# B&R Automation Studio project MotionTestBenchMaster (part 59)

#### LiftMoveMngt_Doser.st
```iecst
ACTION LiftMoveMngt_Doser:

	VAR_DOS_Lift_State.DevicesGeneralAlarm := MMF[205].OUT_DriveFault OR MMF[205].OUT_OverloadFault OR MMF[206].OUT_DriveFault OR
												MMF[206].OUT_OverloadFault OR _205MEF.OUT_Alarm OR _206MEF.OUT_Alarm;

	VAR_DOS_Lift_State.CmdProductionHeight.Sp	:= HMI_PAR_1._215; //[ml]
	VAR_DOS_Lift_State.CmdCipHeight.Sp			:= 145.0; //[ml]

	VAR_DOS_PistonVolume_ml := 145.0; 	(*ml*)  //Max Volume [ml]
	VAR_DOS_PistonVolume_mm := 180.0;	(*mm*)  //Max height of recipe [mm]

	FbLCRLimScal_ml_mm(
	x1 := 0.0, 		(*ml*)
	y1 := 0.0, 		(*mm*)
	x2 := VAR_DOS_PistonVolume_ml, 	(*ml*)
	y2 := VAR_DOS_PistonVolume_mm,	(*mm*)
	);

	FbLCRLimScal_mm_ml(
	x1 := 0.0, 		(*mm*)
	y1 := 0.0, 		(*ml*)
	x2 := VAR_DOS_PistonVolume_mm, 	(*mm*)
	y2 := VAR_DOS_PistonVolume_ml,	(*ml*)
	);

	IF (VAR_DOS_ModePositionRequest AND (VAR_DOS_ModeWait AND NOT COP.DataOut.RcpActive)) THEN
		VAR_DOS_MMF205.SpActual[mm]	:= 200.0; //DEFINE-> Hema Valves "free" - Cam horizontal
		VAR_DOS_MMF206.SpActual[mm]	:= 200.0;
	ELSIF ((VAR_DOS_ModePositionRequest AND (VAR_DOS_ModeProduction OR VAR_DOS_FMDProductionFillerOnly)) OR (HMI_DOS_LiftPosition.Value = 1)) THEN
		VAR_DOS_MMF205.SpActual[ml] := MIN(VAR_DOS_Lift_State.CmdProductionHeight.Sp,VAR_DOS_PistonVolume_ml);
		FbLCRLimScal_ml_mm.x 		:= VAR_DOS_MMF205.SpActual[ml];
		VAR_DOS_MMF205.SpActual[mm]	:= FbLCRLimScal_ml_mm.y;
		VAR_DOS_MMF206.SpActual[mm]	:= 0.0;
	ELSIF ((VAR_DOS_ModePositionRequest AND (VAR_DOS_ModeCip OR VAR_DOS_ModeRinse)) OR (HMI_DOS_LiftPosition.Value = 3)) THEN
		VAR_DOS_MMF205.SpActual[ml] := MIN(VAR_DOS_Lift_State.CmdCipHeight.Sp,VAR_DOS_PistonVolume_ml);
		FbLCRLimScal_ml_mm.x 		:= VAR_DOS_MMF205.SpActual[ml];
		VAR_DOS_MMF205.SpActual[mm]	:= FbLCRLimScal_ml_mm.y;
		VAR_DOS_MMF206.SpActual[mm]	:= 0.0;
	ELSIF ((VAR_DOS_ModePositionRequest AND VAR_DOS_ModeCop AND COP.DataOut.DoserPositioningReq) OR (HMI_DOS_LiftPosition.Value = 2)) THEN
		VAR_DOS_MMF205.SpActual[mm] := 322.0; //High sensor height _215DSF  Define in Test
		VAR_DOS_MMF205.SpActual[ml] := 0;
		VAR_DOS_MMF206.SpActual[mm]	:= 323.0;
	ELSIF HMI_DOS_SS2P[SS2P_DOS_ProbeAdjustment].ON THEN
		VAR_DOS_MMF205.SpActual[mm] := 0.0;
		VAR_DOS_MMF206.SpActual[mm]	:= VAR_DOS_MMF205.SpActual[mm]; //--> Define in Test _205MEF.IN_Delta and _206MEF.IN_Delta
	ELSE
		VAR_DOS_MMF205.SpActual[mm] := 0.0;
		VAR_DOS_MMF205.SpActual[ml] := 0.0;
		VAR_DOS_MMF206.SpActual[mm] := 0.0;
	END_IF

	memset(ADR(VAR_DOS_LiftMMF205SeqMem), 0, SIZEOF(VAR_DOS_LiftMMF205SeqMem));
	memset(ADR(VAR_DOS_LiftMMF206SeqMem), 0, SIZEOF(VAR_DOS_LiftMMF206SeqMem));
	HMI_DOS_PB[PB_DOS_Up].Enable		:= FALSE;
	HMI_DOS_PB[PB_DOS_Down].Enable		:= FALSE;
	_211CPF.IN_AutoCnd 					:= FALSE;
	IF EDGEPOS(VAR_DOS_Lift_State.DevicesGeneralAlarm) THEN
		VAR_DOS_LiftStepMem := VAR_DOS_LiftMoveStep;
	END_IF

	IF EDGENEG(VAR_DOS_ModeWait) OR NOT HMI_DOS_LiftPosition.Enable THEN
		HMI_DOS_LiftPosition.Value := 0;
	END_IF

	IF EDGEPOS(VAR_DOS_FMDPositionRequest) THEN
		VAR_DOS_SeqPositionReached := FALSE;
	END_IF

	//*******************************************************************************************************************************************
	CASE VAR_DOS_LiftMoveStep OF
		DSR_LiftSystemOff:
			HMI_DOS_Lift_State.Sequencer.TextBar[0].IndexNr		:= 0;
			HMI_DOS_Lift_State.Sequencer.TextBar[0].IndexText	:= 0;

			VAR_DOS_LiftMMF205SeqMem.Position.ActualSp	:= VAR_DOS_MMF205.SpActual[ml]; //[ml]

			IF HMI_DOS_SS2P[SS2P_DOS_SelLiftMan].ON THEN
				VAR_DOS_LiftMoveStep := DSR_Manual;
			ELSIF HMI_DOS_SS2P[SS2P_DOS_ProbeAdjustment].ON THEN
				VAR_DOS_LiftMoveStep := DSR_ProbeZeroReq;
			ELSIF (VAR_DOS_ModePositionRequest AND NOT VAR_DOS_SeqPositionReached AND VAR_DOS_ModeWait AND NOT COP.DataOut.RcpActive) THEN
				VAR_DOS_LiftMoveStep := DSR_PosMMF206ToMMF205;
			ELSIF ((VAR_DOS_ModeCop AND COP.DataOut.DoserPositioningReq AND NOT VAR_DOS_SeqPositionReached) OR (EDGEPOS(HMI_DOS_PB[PB_CmdLiftMotorStart].ON) AND HMI_DOS_LiftPosition.Value = 2)) THEN
				VAR_DOS_LiftMoveStep := DSR_PosMMF206ToMMF205;
			ELSIF (((VAR_DOS_ModeProduction OR VAR_DOS_FMDProductionFillerOnly) AND VAR_DOS_ModePositionRequest AND NOT VAR_DOS_SeqPositionReached) OR (EDGEPOS(HMI_DOS_PB[PB_CmdLiftMotorStart].ON) AND HMI_DOS_LiftPosition.Value = 1))THEN
				VAR_DOS_LiftMoveStep := DSR_DosingReq;
			ELSIF (((VAR_DOS_ModeCip OR VAR_DOS_ModeRinse) AND VAR_DOS_ModePositionRequest AND NOT VAR_DOS_SeqPositionReached) OR (EDGEPOS(HMI_DOS_PB[PB_CmdLiftMotorStart].ON) AND HMI_DOS_LiftPosition.Value = 3)) THEN
				VAR_DOS_LiftMoveStep := DSR_DosingReq;
			END_IF

		DSR_ProbeZeroReq:
			HMI_DOS_Lift_State.Sequencer.TextBar[0].IndexNr		:= 1;
			HMI_DOS_Lift_State.Sequencer.TextBar[0].IndexText	:= 1;

			VAR_DOS_LiftMoveStep := DSR_ProbeZeroLowPos;
			IF NOT HMI_DOS_SS2P[SS2P_DOS_ProbeAdjustment].ON THEN
				VAR_DOS_LiftMoveStep := DSR_LiftSystemOff;
			END_IF

		DSR_ProbeZeroLowPos:
			HMI_DOS_Lift_State.Sequencer.TextBar[0].IndexNr		:= 2;
			HMI_DOS_Lift_State.Sequencer.TextBar[0].IndexText	:= 2;

			IF NOT VAR_DOS_Lift_State.DevicesGeneralAlarm THEN

				IF ((VAR_DOS_MMF205.PosActual[mm] <= VAR_DOS_MMF205.SpActual[mm]) OR VAR_DOS_MMF205.SensorLowPos OR (VAR_DOS_MMF205.PosActual[mm] < VAR_DOS_MMF206.PosActual[mm] - 5.0)) THEN
					VAR_DOS_LiftMMF205SeqMem.LiftMotor.Dwn := FALSE;
				ELSIF VAR_DOS_MMF205.SpActual[mm] <= VAR_DOS_MMF205.PosActual[mm] THEN
					VAR_DOS_LiftMMF205SeqMem.LiftMotor.Dwn := TRUE;
				END_IF

				IF ((VAR_DOS_MMF206.PosActual[mm] <= VAR_DOS_MMF206.SpActual[mm]) OR VAR_DOS_MMF206.SensorLowPos OR (VAR_DOS_MMF206.PosActual[mm] <= VAR_DOS_MMF205.PosActual[mm] - VAR_DOS_PistonVolume_mm)) THEN
					VAR_DOS_LiftMMF206SeqMem.LiftMotor.Dwn := FALSE;
				ELSIF ((VAR_DOS_MMF206.PosActual[mm] >= VAR_DOS_MMF205.SpActual[mm]) OR (VAR_DOS_MMF206.PosActual[mm] >= VAR_DOS_MMF206.SpActual[mm] AND VAR_DOS_MMF205.PosReached)) (*mm*)THEN
					VAR_DOS_LiftMMF206SeqMem.LiftMotor.Dwn := TRUE;
				END_IF

				IF VAR_DOS_LiftMMF205SeqMem.LiftMotor.Dwn THEN
					IF VAR_DOS_MMF205.SensorMaxVol THEN
						VAR_DOS_LiftMMF205SeqMem.Sensor.SensorMaxVolWaitOff := TRUE;
					ELSIF NOT VAR_DOS_MMF205.SensorLowPos THEN
						VAR_DOS_LiftMMF205SeqMem.Sensor.SensorLowPosWaitOn := TRUE;
					END_IF
				END_IF

				IF VAR_DOS_LiftMMF206SeqMem.LiftMotor.Dwn THEN
					IF NOT VAR_DOS_MMF206.SensorLowPos THEN
						VAR_DOS_LiftMMF206SeqMem.Sensor.SensorLowPosWaitOn := TRUE;
					END_IF
				END_IF

				IF NOT VAR_DOS_LiftMMF205SeqMem.LiftMotor.Dwn AND NOT VAR_DOS_LiftMMF206SeqMem.LiftMotor.Dwn THEN
					VAR_DOS_LiftMoveStep := DSR_ProbeZeroDisengSensLow;
				END_IF

				IF NOT HMI_DOS_SS2P[SS2P_DOS_ProbeAdjustment].ON THEN
					VAR_DOS_LiftMoveStep := DSR_LiftSystemOff;
				END_IF

			END_IF

		DSR_ProbeZeroDisengSensLow:
			HMI_DOS_Lift_State.Sequencer.TextBar[0].IndexNr		:= 3;
			HMI_DOS_Lift_State.Sequencer.TextBar[0].IndexText	:= 3;

			IF NOT VAR_DOS_Lift_State.DevicesGeneralAlarm THEN
				VAR_DOS_LiftMMF205SeqMem.LiftMotor.Up := VAR_DOS_MMF205.SensorLowPos;
				VAR_DOS_LiftMMF206SeqMem.LiftMotor.Up := VAR_DOS_MMF206.SensorLowPos;

				VAR_DOS_LiftMMF205SeqMem.Sensor.SensorLowPosWaitOff := VAR_DOS_LiftMMF205SeqMem.LiftMotor.Up AND VAR_DOS_MMF205.SensorLowPos;
				VAR_DOS_LiftMMF206SeqMem.Sensor.SensorLowPosWaitOff := VAR_DOS_LiftMMF206SeqMem.LiftMotor.Up AND VAR_DOS_MMF206.SensorLowPos;

				IF NOT VAR_DOS_LiftMMF205SeqMem.LiftMotor.Up AND NOT VAR_DOS_LiftMMF206SeqMem.LiftMotor.Up THEN
					VAR_DOS_LiftMoveStep := DSR_ProbeZeroWaitSensLowPos;
				END_IF

				IF NOT HMI_DOS_SS2P[SS2P_DOS_ProbeAdjustment].ON THEN
					VAR_DOS_LiftMoveStep := DSR_LiftSystemOff;
				END_IF
			END_IF

		DSR_ProbeZeroWaitSensLowPos:
			HMI_DOS_Lift_State.Sequencer.TextBar[0].IndexNr		:= 4;
			HMI_DOS_Lift_State.Sequencer.TextBar[0].IndexText	:= 4;

			IF NOT VAR_DOS_Lift_State.DevicesGeneralAlarm THEN
				VAR_DOS_LiftMMF205SeqMem.LiftMotor.Dwn := NOT VAR_DOS_MMF205.SensorLowPos;
				VAR_DOS_LiftMMF206SeqMem.LiftMotor.Dwn := NOT VAR_DOS_MMF206.SensorLowPos;

				VAR_DOS_LiftMMF205SeqMem.Sensor.SensorLowPosWaitOff := VAR_DOS_LiftMMF205SeqMem.LiftMotor.Up AND NOT VAR_DOS_MMF205.SensorLowPos;
				VAR_DOS_LiftMMF206SeqMem.Sensor.SensorLowPosWaitOff := VAR_DOS_LiftMMF206SeqMem.LiftMotor.Up AND NOT VAR_DOS_MMF206.SensorLowPos;

				IF NOT VAR_DOS_LiftMMF205SeqMem.LiftMotor.Dwn AND NOT VAR_DOS_LiftMMF206SeqMem.LiftMotor.Dwn THEN
					VAR_DOS_MMF205.PosValid := FALSE;
					VAR_DOS_MMF206.PosValid := FALSE;
					Delta_205MEF			:= 0.0;
					Delta_206MEF			:= 0.0;
					VAR_DOS_LiftMoveStep	:= DSR_ProbeZeroDone;
				END_IF
			END_IF

			IF NOT HMI_DOS_SS2P[SS2P_DOS_ProbeAdjustment].ON THEN
				VAR_DOS_LiftMoveStep := DSR_LiftSystemOff;
			END_IF

		DSR_ProbeZeroDone:
			HMI_DOS_Lift_State.Sequencer.TextBar[0].IndexNr		:= 5;
			HMI_DOS_Lift_State.Sequencer.TextBar[0].IndexText	:= 5;

			IF NOT VAR_DOS_Lift_State.DevicesGeneralAlarm THEN
				IF NOT VAR_DOS_MMF205.PosValid THEN
					Delta_205MEF			:= -(_205MEF.OUT_ActValue + Delta_205MEF) + 0.5;
					VAR_DOS_MMF205.PosValid := TRUE;
				END_IF

				IF NOT VAR_DOS_MMF206.PosValid THEN
					Delta_206MEF 		:= -(_206MEF.OUT_ActValue + Delta_206MEF) + 0.5;
					VAR_DOS_MMF206.PosValid := TRUE;
				END_IF
			END_IF

			IF VAR_DOS_MMF205.PosValid AND VAR_DOS_MMF206.PosValid THEN
				HMI_DOS_SS2P[SS2P_DOS_ProbeAdjustment].ON := FALSE;
				VAR_DOS_LiftMoveStep					  := DSR_LiftSystemOff;
			END_IF

		DSR_PosMMF206ToMMF205:
			HMI_DOS_Lift_State.Sequencer.TextBar[0].IndexNr		:= 10;
			HMI_DOS_Lift_State.Sequencer.TextBar[0].IndexText	:= 10;
			VAR_DOS_LiftMMF205SeqMem.Position.ActualSp	:= VAR_DOS_MMF205.SpActual[ml]; //[ml]
			VAR_DOS_SeqPositionReached	:= FALSE;

			IF NOT VAR_DOS_Lift_State.DevicesGeneralAlarm THEN
				IF VAR_DOS_ModeCop THEN
					VAR_DOS_LiftMMF206SeqMem.LiftMotor.Up := (VAR_DOS_MMF206.PosActual[mm] < VAR_DOS_MMF205.PosActual[mm]);
					IF NOT VAR_DOS_LiftMMF206SeqMem.LiftMotor.Up THEN
						VAR_DOS_LiftMoveStep := DSR_UpMMF205andMMF206;
					END_IF
				ELSIF VAR_DOS_MMF205.SpActual[mm] >= VAR_DOS_MMF205.PosActual[mm] THEN
					VAR_DOS_LiftMMF206SeqMem.LiftMotor.Up := VAR_DOS_MMF206.PosActual[mm] < VAR_DOS_MMF205.PosActual[mm];
					IF NOT VAR_DOS_LiftMMF206SeqMem.LiftMotor.Up THEN
						VAR_DOS_LiftMoveStep := DSR_UpMMF205andMMF206;
					END_IF
				END_IF
			ELSE
				VAR_DOS_LiftMoveStep := DSR_Fault;
			END_IF

		DSR_UpMMF205andMMF206:
			HMI_DOS_Lift_State.Sequencer.TextBar[0].IndexNr		:= 11;
			HMI_DOS_Lift_State.Sequencer.TextBar[0].IndexText	:= 11;

			VAR_DOS_LiftMMF205SeqMem.Position.ActualSp	:= VAR_DOS_MMF205.SpActual[ml]; //[ml]

			IF EDGEPOS(HMI_DOS_PB[PB_CmdLiftMotorStop].ON) THEN
				VAR_DOS_LiftMoveStep := DSR_LiftSystemOff;
			END_IF

			IF NOT VAR_DOS_Lift_State.DevicesGeneralAlarm THEN

				IF ((VAR_DOS_MMF205.PosActual[mm] > VAR_DOS_MMF205.SpActual[mm]) OR VAR_DOS_MMF205.SensorHighPos OR (VAR_DOS_MMF205.PosActual[mm] > VAR_DOS_MMF206.PosActual[mm] + VAR_DOS_PistonVolume_mm)) THEN
					VAR_DOS_LiftMMF205SeqMem.LiftMotor.Up := FALSE;
				ELSIF VAR_DOS_MMF205.SpActual[mm] >= VAR_DOS_MMF205.PosActual[mm] THEN
					VAR_DOS_LiftMMF205SeqMem.LiftMotor.Up := TRUE;
				END_IF

				IF ((VAR_DOS_MMF206.PosActual[mm] > VAR_DOS_MMF206.SpActual[mm]) OR VAR_DOS_MMF206.SensorHighPos OR (VAR_DOS_MMF206.PosActual[mm] > VAR_DOS_MMF205.PosActual[mm] + 5.0)) THEN
					VAR_DOS_LiftMMF206SeqMem.LiftMotor.Up := FALSE;
				ELSIF VAR_DOS_MMF206.PosActual[mm] <= VAR_DOS_MMF206.SpActual[mm] THEN //CHECK
					VAR_DOS_LiftMMF206SeqMem.LiftMotor.Up := TRUE;
				END_IF

				IF NOT VAR_DOS_LiftMMF205SeqMem.LiftMotor.Up THEN
					VAR_DOS_MMF205.PosReached := TRUE;
				ELSE
					VAR_DOS_MMF205.PosReached := FALSE;
				END_IF

				IF NOT VAR_DOS_LiftMMF206SeqMem.LiftMotor.Up THEN
					VAR_DOS_MMF206.PosReached := TRUE;
				ELSE
					VAR_DOS_MMF206.PosReached := FALSE;
				END_IF

				IF ((VAR_DOS_ModeCop AND COP.DataOut.DoserPositioningReq) OR (VAR_DOS_ModeWait AND (HMI_DOS_LiftPosition.Value = 2))) THEN
					IF VAR_DOS_MMF206.PosReached AND VAR_DOS_MMF205.PosReached AND VAR_DOS_MMF205.SensorHighPos AND VAR_DOS_MMF206.SensorHighPos THEN
						VAR_DOS_LiftMoveStep := DSR_CopPosReached;
					END_IF
				ELSE
					VAR_DOS_LiftMoveStep := DSR_LiftSystemOff;
				END_IF
			ELSE
				VAR_DOS_LiftMoveStep := DSR_Fault;
			END_IF

		DSR_DwnMMF205andMMF206:
			HMI_DOS_Lift_State.Sequencer.TextBar[0].IndexNr		:= 12;
			HMI_DOS_Lift_State.Sequencer.TextBar[0].IndexText	:= 12;

			VAR_DOS_LiftMMF205SeqMem.Position.ActualSp	:= VAR_DOS_MMF205.SpActual[ml]; //[ml]

			IF EDGEPOS(HMI_DOS_PB[PB_CmdLiftMotorStop].ON) THEN
				VAR_DOS_LiftMoveStep := DSR_LiftSystemOff;
			END_IF

			IF NOT VAR_DOS_Lift_State.DevicesGeneralAlarm THEN

				IF ((VAR_DOS_MMF205.PosActual[mm] < VAR_DOS_MMF205.SpActual[mm]) OR VAR_DOS_MMF205.SensorLowPos OR (VAR_DOS_MMF205.PosActual[mm] < VAR_DOS_MMF206.PosActual[mm] - 5.0)) THEN
					VAR_DOS_LiftMMF205SeqMem.LiftMotor.Dwn := FALSE;
				ELSIF VAR_DOS_MMF205.SpActual[mm] <= VAR_DOS_MMF205.PosActual[mm] THEN
					VAR_DOS_LiftMMF205SeqMem.LiftMotor.Dwn := TRUE;
				END_IF

				IF ((VAR_DOS_MMF206.PosActual[mm] < VAR_DOS_MMF206.SpActual[mm]) OR VAR_DOS_MMF206.SensorLowPos OR (VAR_DOS_MMF206.PosActual[mm] <= VAR_DOS_MMF205.PosActual[mm] - VAR_DOS_PistonVolume_mm)) THEN
					VAR_DOS_LiftMMF206SeqMem.LiftMotor.Dwn := FALSE;
				ELSIF ((VAR_DOS_MMF206.PosActual[mm] >= VAR_DOS_MMF205.SpActual[mm]) OR (VAR_DOS_MMF206.PosActual[mm] >= VAR_DOS_MMF206.SpActual[mm])) (*mm*)THEN
					VAR_DOS_LiftMMF206SeqMem.LiftMotor.Dwn := TRUE;
					END_IF

				IF NOT VAR_DOS_LiftMMF205SeqMem.LiftMotor.Dwn THEN
					VAR_DOS_MMF205.PosReached := TRUE;
				ELSE
					VAR_DOS_MMF205.PosReached := FALSE;
				END_IF

				IF NOT VAR_DOS_LiftMMF206SeqMem.LiftMotor.Dwn THEN
					VAR_DOS_MMF206.PosReached := TRUE;
				ELSE
					VAR_DOS_MMF206.PosReached := FALSE;
				END_IF

				IF (VAR_DOS_ModeCop AND COP.DataOut.DoserPositioningReq) OR (VAR_DOS_ModeWait AND HMI_DOS_LiftPosition.Value = 2) THEN
					IF VAR_DOS_MMF206.PosReached AND VAR_DOS_MMF206.SensorHighPos AND VAR_DOS_MMF205.SensorHighPos THEN
						VAR_DOS_LiftMoveStep := DSR_CopPosReached;
					END_IF
				ELSIF (VAR_DOS_ModeProduction OR VAR_DOS_FMDProductionFillerOnly) OR (VAR_DOS_ModeWait AND HMI_DOS_LiftPosition.Value = 1)THEN
					IF VAR_DOS_MMF206.PosReached AND VAR_DOS_MMF206.SensorLowPos THEN
						VAR_DOS_LiftMoveStep := DSR_DosingActive;
					END_IF
				ELSIF (VAR_DOS_ModeCip OR VAR_DOS_ModeRinse) OR (VAR_DOS_ModeWait AND HMI_DOS_LiftPosition.Value = 3) THEN
					IF VAR_DOS_MMF206.PosReached AND VAR_DOS_MMF206.SensorLowPos THEN
						VAR_DOS_LiftMoveStep := DSR_DosingActive;
					END_IF
				ELSE
					VAR_DOS_LiftMoveStep := DSR_LiftSystemOff;
				END_IF
			ELSE
				VAR_DOS_LiftMoveStep := DSR_Fault;
			END_IF

		DSR_CopPosReached:
			HMI_DOS_Lift_State.Sequencer.TextBar[0].IndexNr		:= 6;
			HMI_DOS_Lift_State.Sequencer.TextBar[0].IndexText	:= 6;

			VAR_DOS_LiftMMF205SeqMem.Position.ActualSp	:= VAR_DOS_MMF205.SpActual[ml]; //[ml]

			_211CPF.IN_AutoCnd := COP.DataOut.DoserPositioningReq AND VAR_DOS_MMF205.SensorHighPos AND VAR_DOS_MMF206.SensorHighPos;

			VAR_DOS_SeqPositionReached := _210DSX.OUT;

			IF NOT COP.DataOut.DoserPositioningReq AND _211DSX.OUT THEN
				VAR_DOS_LiftMoveStep := DSR_LiftSystemOff;
			END_IF

		DSR_DosingReq:
			HMI_DOS_Lift_State.Sequencer.TextBar[0].IndexNr		:= 7;
			IF VAR_DOS_ModeCip THEN
				HMI_DOS_Lift_State.Sequencer.TextBar[0].IndexText	:= 15;//CIP
			ELSIF VAR_DOS_ModeProduction THEN
				HMI_DOS_Lift_State.Sequencer.TextBar[0].IndexText	:= 7;//PRODUCTION
			END_IF
			VAR_DOS_LiftMMF205SeqMem.Position.ActualSp	:= VAR_DOS_MMF205.SpActual[ml]; //[ml]
			VAR_DOS_SeqPositionReached	:= FALSE;

			IF NOT VAR_DOS_MMF206.SensorLowPos THEN
				VAR_DOS_LiftMoveStep := DSR_DwnMMF205andMMF206;
			ELSE
				VAR_DOS_LiftMoveStep := DSR_DosingActive;
			END_IF

		DSR_DosingActive:
			HMI_DOS_Lift_State.Sequencer.TextBar[0].IndexNr		:= 8;
			HMI_DOS_Lift_State.Sequencer.TextBar[0].IndexText	:= 8;

			VAR_DOS_LiftMMF205SeqMem.Position.ActualSp	:= VAR_DOS_MMF205.SpActual[ml]; //[ml]

			IF EDGEPOS(HMI_DOS_PB[PB_CmdLiftMotorStop].ON) THEN
				VAR_DOS_LiftMoveStep := DSR_LiftSystemOff;
			END_IF

			IF NOT VAR_DOS_Lift_State.DevicesGeneralAlarm THEN

				IF ((VAR_DOS_MMF205.PosActual[mm] > VAR_DOS_MMF205.SpActual[mm]) OR VAR_DOS_MMF205.SensorHighPos OR VAR_DOS_MMF205.SensorMaxVol OR (VAR_DOS_MMF205.PosActual[mm] > VAR_DOS_MMF206.PosActual[mm] + VAR_DOS_PistonVolume_mm)) THEN
					VAR_DOS_LiftMMF205SeqMem.LiftMotor.Up := FALSE;
				ELSIF VAR_DOS_MMF205.SpActual[mm] - 0.5 >= VAR_DOS_MMF205.PosActual[mm] THEN
					VAR_DOS_LiftMMF205SeqMem.LiftMotor.Up := TRUE;
				END_IF

				IF ((VAR_DOS_MMF205.PosActual[mm] < VAR_DOS_MMF205.SpActual[mm]) OR VAR_DOS_MMF205.SensorLowPos) THEN
					VAR_DOS_LiftMMF205SeqMem.LiftMotor.Dwn := FALSE;
				ELSIF VAR_DOS_MMF205.SpActual[mm] + 0.5 <= VAR_DOS_MMF205.PosActual[mm] THEN
					VAR_DOS_LiftMMF205SeqMem.LiftMotor.Dwn := TRUE;
				END_IF

				IF (NOT VAR_DOS_LiftMMF205SeqMem.LiftMotor.Up AND NOT VAR_DOS_LiftMMF205SeqMem.LiftMotor.Dwn) THEN
					VAR_DOS_MMF205.PosReached := TRUE;
				ELSE
					VAR_DOS_MMF205.PosReached := FALSE;
				END_IF

				VAR_DOS_MMF206.PosReached	:= VAR_DOS_MMF206.SensorLowPos;

				VAR_DOS_SeqPositionReached	:= VAR_DOS_MMF205.PosReached AND VAR_DOS_MMF206.PosReached;

				IF VAR_DOS_SeqPositionReached THEN
					VAR_DOS_LiftMoveStep := DSR_LiftSystemOff;
				END_IF
			ELSE
				VAR_DOS_LiftMoveStep := DSR_Fault;
			END_IF

		DSR_Manual:
			HMI_DOS_Lift_State.Sequencer.TextBar[0].IndexNr		:= 9;
			HMI_DOS_Lift_State.Sequencer.TextBar[0].IndexText	:= 9;

			VAR_DOS_LiftMMF205SeqMem.Position.ActualSp	:= VAR_DOS_MMF205.SpActual[ml]; //[ml]

			IF NOT VAR_DOS_Lift_State.DevicesGeneralAlarm THEN
				IF HMI_DOS_SS2P[SS2P_DOS_ManualMMF205].LampON AND NOT VAR_DOS_MMF205.SensorHighPos AND VAR_DOS_MMF205.PosActual[mm] <= VAR_DOS_MMF206.PosActual[mm] + VAR_DOS_PistonVolume_mm THEN
					HMI_DOS_PB[PB_DOS_Up].Enable := TRUE;
					VAR_DOS_LiftMMF205SeqMem.LiftMotor.Up := HMI_DOS_PB[PB_DOS_Up].LampON;
				ELSIF HMI_DOS_SS2P[SS2P_DOS_ManualMMF206].LampON AND NOT VAR_DOS_MMF206.SensorHighPos AND VAR_DOS_MMF206.PosActual[mm] <= VAR_DOS_MMF205.PosActual[mm] THEN
					HMI_DOS_PB[PB_DOS_Up].Enable := TRUE;
					VAR_DOS_LiftMMF206SeqMem.LiftMotor.Up := HMI_DOS_PB[PB_DOS_Up].LampON;
				END_IF

				IF HMI_DOS_SS2P[SS2P_DOS_ManualMMF205].LampON AND NOT VAR_DOS_MMF205.SensorLowPos AND VAR_DOS_MMF205.PosActual[mm] >= VAR_DOS_MMF206.PosActual[mm] - 10.0 THEN
					HMI_DOS_PB[PB_DOS_Down].Enable := TRUE;
					VAR_DOS_LiftMMF205SeqMem.LiftMotor.Dwn := HMI_DOS_PB[PB_DOS_Down].LampON;
				ELSIF HMI_DOS_SS2P[SS2P_DOS_ManualMMF206].LampON AND NOT VAR_DOS_MMF206.SensorLowPos AND VAR_DOS_MMF206.PosActual[mm] >= VAR_DOS_MMF205.PosActual[mm] - VAR_DOS_PistonVolume_mm THEN
					HMI_DOS_PB[PB_DOS_Down].Enable := TRUE;
					VAR_DOS_LiftMMF206SeqMem.LiftMotor.Dwn := HMI_DOS_PB[PB_DOS_Down].LampON;
				END_IF
			END_IF

			IF NOT HMI_DOS_SS2P[SS2P_DOS_SelLiftMan].ON THEN
				VAR_DOS_LiftMoveStep := DSR_LiftSystemOff;
			END_IF

		DSR_Fault:
			HMI_DOS_Lift_State.Sequencer.TextBar[0].IndexNr	:= 13;
			HMI_DOS_Lift_State.Sequencer.TextBar[0].IndexText 	:= 13;

			VAR_DOS_SeqPositionReached	:= FALSE;

			VAR_DOS_LiftMMF205SeqMem.Position.ActualSp	:= VAR_DOS_MMF205.SpActual[ml] * BOOL_TO_REAL(VAR_DOS_ModePositionRequest);
			IF NOT VAR_DOS_Lift_State.DevicesGeneralAlarm THEN
				VAR_DOS_LiftMoveStep := VAR_DOS_LiftStepMem;
			END_IF

	END_CASE
	//******************************************************************************************************************************************

	MMF[205].IN_AutoCnd		:= (VAR_DOS_LiftMMF205SeqMem.LiftMotor.Up AND NOT VAR_DOS_MMF205.SensorHighPos) OR
	(VAR_DOS_LiftMMF205SeqMem.LiftMotor.Dwn AND NOT VAR_DOS_MMF205.SensorLowPos);
	MMF[205].IN_Reverse		:= VAR_DOS_LiftMMF205SeqMem.LiftMotor.Dwn AND MMF[205].IN_AutoCnd;

	MMF[206].IN_AutoCnd		:= (VAR_DOS_LiftMMF206SeqMem.LiftMotor.Up AND NOT VAR_DOS_MMF206.SensorHighPos) OR
	(VAR_DOS_LiftMMF206SeqMem.LiftMotor.Dwn AND NOT VAR_DOS_MMF206.SensorLowPos);
	MMF[206].IN_Reverse		:= VAR_DOS_LiftMMF206SeqMem.LiftMotor.Dwn AND MMF[206].IN_AutoCnd;

	_215DSF.IN_WaitOn	:= VAR_DOS_LiftMMF205SeqMem.Sensor.SensorHighPosWaitOn;
	_215DSF.IN_WaitOff	:= VAR_DOS_LiftMMF205SeqMem.Sensor.SensorHighPosWaitOff;

	_216DSF.IN_WaitOn	:= VAR_DOS_LiftMMF206SeqMem.Sensor.SensorHighPosWaitOn;
	_216DSF.IN_WaitOff	:= VAR_DOS_LiftMMF206SeqMem.Sensor.SensorHighPosWaitOff;
	_217DSF.IN_WaitOn	:= VAR_DOS_LiftMMF206SeqMem.Sensor.SensorLowPosWaitOn;
	_217DSF.IN_WaitOff	:= VAR_DOS_LiftMMF206SeqMem.Sensor.SensorLowPosWaitOff;

	VAR_DOS_MMF205.SensorHighPos := _215DSF.OUT AND NOT _212DSF.OUT AND NOT _213DSF.OUT;
	VAR_DOS_MMF205.SensorMaxVol  := NOT _212DSF.OUT AND _213DSF.OUT;
	VAR_DOS_MMF205.SensorLowPos	 := NOT _213DSF.OUT AND NOT _215DSF.OUT AND _212DSF.OUT;
	VAR_DOS_MMF205.PosActual[mm] := _205MEF.OUT_ActValue;
	FbLCRLimScal_mm_ml.x		 := VAR_DOS_MMF205.PosActual[mm];
	VAR_DOS_MMF205.PosActual[ml] := FbLCRLimScal_mm_ml.y;

	VAR_DOS_MMF206.SensorHighPos := _216DSF.OUT AND NOT _217DSF.OUT;
	VAR_DOS_MMF206.SensorLowPos  := _217DSF.OUT AND NOT _216DSF.OUT;
	VAR_DOS_MMF206.PosActual[mm] := _206MEF.OUT_ActValue;

	IF _205MEF.OUT_Alarm AND MMF[205].OUT_InOperation THEN
		VAR_DOS_MMF205.PosValid := FALSE;
	END_IF
	IF _206MEF.OUT_Alarm AND MMF[206].OUT_InOperation THEN
		VAR_DOS_MMF206.PosValid := FALSE;
	END_IF

	END_ACTION
```

#### DOS_DataOut.st
```iecst
ACTION DOS_DataOut:

	//SEQUENCE
	DOS.DataOut.WaitMode		:= VAR_DOS_ModeWait;
	DOS.DataOut.ProdMode		:= VAR_DOS_ModeProduction;
	DOS.DataOut.CipMode 		:= VAR_DOS_ModeCip;
	DOS.DataOut.RinseMode		:= VAR_DOS_ModeRinse;
	DOS.DataOut.CopMode			:= VAR_DOS_ModeCop AND VAR_DOS_SeqPositionReached;
	DOS.DataOut.DrainMode		:= VAR_DOS_ModeDrain;
	DOS.DataOut.CopAfterCipReq  := VAR_DOS_SEQ.Mem.CopAfterCipRequest;
	DOS.DataOut.CopRunning		:= VAR_DOS_StepCopRunning;

	//SIGNALS INTERCHANGE
	DOS.DataOut.FillingProd		:= VAR_DOS_StepProdProducing OR VAR_DOS_StepProdEndProduction;
	DOS.DataOut.CommandToValve	:= VAR_DOS_SEQ.Mem.ValveOpening OR COP.DataOut.RcpActive;
	DOS.DataOut.ProductRequest	:= VAR_DOS_SEQ.ITC.PROD_ProductRequest; //PULP REQ
	DOS.DataOut.ProductionEnd	:= VAR_DOS_SEQ.ITC.PROD_EndProductionCompleted;
	DOS.DataOut.ReadyForHeating := VAR_DOS_SEQ.ITC.PROD_ReadyForHeating; //HOT WATER REQ
	DOS.DataOut.DoserInTemperature := TTJ[203].OUT_SpReached;
	DOS.DataOut.DoserFull		:= LTJ[203].OUT_SpReached AND VAR_DOS_StepProdHeating; //ONLY IN START UP ?
	DOS.DataOut.AVJ201Open		:= AVJ[201].OUT_OpenedFiltered;
	DOS.DataOut.DoserEmpty		:= VAR_DOS_TankEmpted;
	DOS.DataOut.RecoveryEnd		:= VAR_DOS_SEQ.ITC.PROD_ProductRecoveryEnd;

	DOS.DataOut.CipConditionOk	:= VAR_DOS_ModeCip AND VAR_DOS_SeqPositionReached AND NOT VAR_DOS_SeqCipStopAlarm AND TTJ[203].OUT_SpReached; //CIP SOLUT REQ AND CIP SOLUTION RETURN
	DOS.DataOut.CipSolutionReq	:= VAR_DOS_SEQ.ITC.CIP_CleaningRequest;
	DOS.DataOut.CipAlarm		:= VAR_DOS_SeqCipStopAlarm; //VALUTA
	DOS.DataOut.CipRecovery		:= VAR_DOS_StepCipRecovery AND IO_AVJ[216].DI_Opened AND AVJ[217].OUT (*AND IO_AVJ[218].DI_Opened*) AND PPJ[202].OUT_InOperation;
	DOS.DataOut.CipRecoveryEnd  := VAR_DOS_SEQ.ITC.CIP_ChangeEnded;
	DOS.DataOut.CipSystemFlooded := VAR_DOS_SEQ.ITC.CIP_FloodingEnded;
	DOS.DataOut.CipDrainEnd		:= VAR_DOS_SEQ.ITC.CIP_DrainEnded;
	DOS.DataOut.CipLevelReached := LTJ[203].OUT_SpReached AND VAR_DOS_ModeCip; //Allo step 73 A2 aspetta che tutti i partner siano a livelloCIP e poi chiude tutto in loop

	DOS.DataOut.RinseReq		:= VAR_DOS_SEQ.ITC.CIP_RinseRunning;
	DOS.DataOut.RinseEnd		:= VAR_DOS_SEQ.ITC.CIP_RinseEnded;
	DOS.DataOut.RinseAfterProdReq := VAR_DOS_SEQ.ITC.PROD_WaterRequestAfterProd;
	DOS.DataOut.RinseAfterProdEnd := VAR_DOS_SEQ.ITC.CIP_RinseEnded;

	DOS.DataOut.EjectionRequest	:= VAR_DOS_RejectExpulsionRequest;
	DOS.DataOut.HotWaterReq		:= VAR_DOS_StepCipDraining; //At the end of the CIP, rinse of hot water

	DOS.DataOut.NecessaryBottleEndProd := VAR_DOS_ProdEndNecessaryBottle;

	//FIX SPEED
	DOS.DataOut.FixSpeedRequest := (VAR_DOS_ModeCip AND NOT TNK.DataOut.CipMode) OR VAR_DOS_ModeCop OR (VAR_DOS_ModeRinse AND NOT TNK.DataOut.RinseMode);

	IF VAR_DOS_ModeCip OR VAR_DOS_ModeRinse THEN
		DOS.DataOut.FixSpeedValue := HMI_PAM_3._631;
	ELSIF VAR_DOS_FMDCop THEN
		DOS.DataOut.FixSpeedValue := HMI_PAM_3._632;
	END_IF

	//MOTION
	DOS.DataOut.MachineStart			:= VAR_DOS_SEQ.Mem.MachineStart;
	DOS.DataOut.MachineStop				:= VAR_DOS_SEQ.Mem.MachineStop;
	DOS.DataOut.DoserExcluded 			:= VAR_DOS_MemDoserByPassed;
	DOS.DataOut.DoserIncluded			:= VAR_DOS_MemDoserIncluded;
	DOS.DataOut.ByPassed				:= GNS.DataOut.DosByPassed;
	DOS.DataOut.PhasingWithDos			:= VAR_DOS_PhasingWithDos;
	DOS.DataOut.PhasingWithoutDos			:= VAR_DOS_PhasingWithoutDos;

	IF OPS.DataOut.FlrModeSelectorAdjustment AND NOT MNM.DataOut.MachineRunning THEN //machine running non so se serve
		DOS.DataOut.AxisDisableRequest		:= FALSE;
		DOS.DataOut.RunOnlyHemaAxisRequest := FALSE;
	ELSE
		DOS.DataOut.AxisDisableRequest		:= VAR_DOS_MemDoserAxisOff;
		DOS.DataOut.AxisEnableRequest		:= VAR_DOS_MemDoserAxisOn;
		DOS.DataOut.RunOnlyHemaAxisRequest  := VAR_DOS_MemFillerAxisOffReq AND NOT TNK.DataOut.StartCipRinser;
		DOS.DataOut.RunRinserHemaAxisRequest := VAR_DOS_MemFillerAxisOffReq AND RNS.DataOut.RunWithHemaReq;
	END_IF

	DOS.DataOut.StepCounterRequest		:= VAR_DOS_SEQ.Mem.LapsCounter;

	DOS.DataOut.PositionReached 		:= VAR_DOS_SeqPositionReached;

	//FILLER SELECTION ENABLE
	DOS.DataOut.FillerProdStartEnable	:= VAR_DOS_ModeWait OR VAR_DOS_ModeProduction;
	DOS.DataOut.FillerCipStartEnable	:= VAR_DOS_ModeWait OR (VAR_DOS_ModeCip AND VAR_DOS_StepCipFillerStartEnable);
	DOS.DataOut.FillerRinseStartEnable	:= VAR_DOS_ModeWait OR VAR_DOS_ModeRinse; //VALUTARE: AND NOT VAR_DOS_StepRinseInExecution)
END_ACTION
```

#### DOS_DataOutFlavor.st
```iecst
ACTION DOS_DataOutFlavor:
	//FLAVOR DOSER
	DOS.DataOut.ProdMode 	:= REAL_TO_BOOL(HMI_PAR_1._005) AND TNK.DataOut.ProdMode;
	DOS.DataOut.CipMode 	:= DosFlr.CipReady OR DosFlr.CipRunning;
	DOS.DataOut.AromePodReq := REAL_TO_BOOL(HMI_PAR_1._005) AND TNK.DataOut.ProdMode;
	DOS.DataOut.MachineStart := DosFlr.RotationRequest;

	IF DOS.DataOut.AromePodReq AND NOT ALR[3100].Active AND DosFlr.PrimingCycleProgress THEN
		DOS.DataOut.FixSpeedRequest 		:= TRUE;
		DOS.DataOut.FixSpeedValue 			:= CFG_MC.Movements.MachineMaxSpeed;
	ELSIF DosFlr.RotationRequest AND NOT ALR[3100].Active AND DOS.DataOut.CipMode THEN
		DOS.DataOut.FixSpeedRequest 		:= TRUE;
		DOS.DataOut.FixSpeedValue 			:= MIN(20000, CFG_MC.Movements.MachineMaxSpeed *0.7);
	ELSIF DosFlr.SampleCycleInProgress THEN
		DOS.DataOut.FixSpeedRequest		 	:= TRUE;
		DOS.DataOut.FixSpeedValue 			:= MIN(10000, CFG_MC.Movements.MachineMaxSpeed *0.5);
	ELSE
		DOS.DataOut.FixSpeedRequest		 	:= FALSE;
		DOS.DataOut.FixSpeedValue 			:= 0;
	END_IF
END_ACTION
```

#### DOS_HMI.st
```iecst
ACTION DOS_HMI:
	VAR_DOS_MemPBStart			:= FALSE;
	VAR_DOS_MemPBStop			:= FALSE;
	VAR_DOS_MemPBAbort			:= FALSE;
	VAR_DOS_MemPBSkipForward	:= FALSE;

	IF NOT HMI_SS2P[SS2P_HMI_SelEnable].ON THEN
		HMI_DOS_SS2P[SS2P_DOS_SelLiftMan].ON := FALSE;
	END_IF

	//SS2P
	//MODE MAN/AUTO
	VAR_DOS_SS2PSelectionEnable := VAR_DOS_ModeWait AND SFT.DataOut.MachineEmpty;

	HMI_DOS_SS2P[SS2P_DOS_ProbeAdjustment].Visibility		:= _205MEF.IN_ConfigPresent AND _206MEF.IN_ConfigPresent;
	HMI_DOS_SS2P[SS2P_DOS_ProbeAdjustment].Enable			:= HMI_SS2P[SS2P_HMI_SelEnable].ON AND VAR_DOS_ModeWait AND OPS.DataOut.FlrModeSelectorAdjustment AND NOT (VAR_DOS_LiftMoveStep = DSR_ProbeZeroWaitSensLowPos) AND NOT (VAR_DOS_LiftMoveStep = DSR_ProbeZeroDone) AND NOT HMI_DOS_SS2P[SS2P_DOS_SelLiftMan].ON;
	HMI_DOS_SS2P[SS2P_DOS_ProbeAdjustment].LampON			:= HMI_DOS_SS2P[SS2P_DOS_ProbeAdjustment].ON AND HMI_DOS_SS2P[SS2P_DOS_ProbeAdjustment].Enable;

	IF EDGEPOS(VAR_DOS_MemDoserByPassed) THEN
		HMI_DOS_SS2P[SS2P_DOS_CamDosByPass].ON := FALSE;
	END_IF
	HMI_DOS_SS2P[SS2P_DOS_CamDosByPass].Visibility			:= GNS.DataOut.DosByPassConfigured AND NOT CFG_Par.Machine.Type.SRMA;
	HMI_DOS_SS2P[SS2P_DOS_CamDosByPass].Enable				:= HMI_SS2P[SS2P_HMI_SelEnable].ON AND VAR_DOS_ModeWait AND TNK.DataOut.Wait AND NOT MNM.DataOut.MachineRunning AND NOT VAR_DOS_MemDoserByPassed;
	HMI_DOS_SS2P[SS2P_DOS_CamDosByPass].LampON				:= HMI_DOS_SS2P[SS2P_DOS_CamDosByPass].ON OR VAR_DOS_MemDoserByPassed;

	IF EDGEPOS(VAR_DOS_MemDoserIncluded) THEN
		HMI_DOS_SS2P[SS2P_DOS_CamDosInclusion].ON := FALSE;
	END_IF
	HMI_DOS_SS2P[SS2P_DOS_CamDosInclusion].Visibility		:= GNS.DataOut.DosByPassConfigured AND NOT CFG_Par.Machine.Type.SRMA;
	HMI_DOS_SS2P[SS2P_DOS_CamDosInclusion].Enable			:= HMI_SS2P[SS2P_HMI_SelEnable].ON AND VAR_DOS_ModeWait  AND TNK.DataOut.Wait AND NOT MNM.DataOut.MachineRunning AND NOT VAR_DOS_MemDoserIncluded;
	HMI_DOS_SS2P[SS2P_DOS_CamDosInclusion].LampON			:= HMI_DOS_SS2P[SS2P_DOS_CamDosInclusion].ON OR VAR_DOS_MemDoserIncluded;

	HMI_DOS_SS2P[SS2P_DOS_SelLiftMan].Visibility		:= TRUE;
	HMI_DOS_SS2P[SS2P_DOS_SelLiftMan].Enable			:= HMI_SS2P[SS2P_HMI_SelEnable].ON AND VAR_DOS_ModeWait AND HMI_DOS_LiftPosition.Value = 0 AND OPS.DataOut.FlrModeSelectorAdjustment AND NOT HMI_DOS_SS2P[SS2P_DOS_ProbeAdjustment].ON;
	HMI_DOS_SS2P[SS2P_DOS_SelLiftMan].LampON			:= HMI_DOS_SS2P[SS2P_DOS_SelLiftMan].ON AND HMI_DOS_SS2P[SS2P_DOS_SelLiftMan].Enable;

	//SS2P DOSER LIFTING
	HMI_DOS_SS2P[SS2P_DOS_ManualMMF206].Visibility	:= TRUE;
	HMI_DOS_SS2P[SS2P_DOS_ManualMMF206].Enable		:= HMI_SS2P[SS2P_HMI_SelEnable].ON AND OPS.DataOut.FlrModeSelectorAdjustment AND OPS.DataOut.FlrDoorsOk	AND OPS.DataOut.EmergencyOk AND HMI_DOS_SS2P[SS2P_DOS_SelLiftMan].ON AND VAR_DOS_ModeWait AND NOT HMI_DOS_SS2P[SS2P_DOS_ManualMMF205].LampON;
	HMI_DOS_SS2P[SS2P_DOS_ManualMMF206].LampON		:= HMI_DOS_SS2P[SS2P_DOS_ManualMMF206].ON AND HMI_DOS_SS2P[SS2P_DOS_ManualMMF206].Enable;

	//SS2P DOSER LIFTING
	HMI_DOS_SS2P[SS2P_DOS_ManualMMF205].Visibility	:= TRUE;
	HMI_DOS_SS2P[SS2P_DOS_ManualMMF205].Enable		:= HMI_SS2P[SS2P_HMI_SelEnable].ON AND OPS.DataOut.FlrModeSelectorAdjustment AND OPS.DataOut.FlrDoorsOk	AND OPS.DataOut.EmergencyOk AND HMI_DOS_SS2P[SS2P_DOS_SelLiftMan].ON AND VAR_DOS_ModeWait AND NOT HMI_DOS_SS2P[SS2P_DOS_ManualMMF206].LampON;
	HMI_DOS_SS2P[SS2P_DOS_ManualMMF205].LampON		:= HMI_DOS_SS2P[SS2P_DOS_ManualMMF205].ON AND HMI_DOS_SS2P[SS2P_DOS_ManualMMF205].Enable;

	//SS2P DOSER PROD
	HMI_DOS_SS2P[SS2P_DOS_ModeProdFast].Visibility	:= TRUE;
	HMI_DOS_SS2P[SS2P_DOS_ModeProdFast].Enable		:= VAR_DOS_SS2PSelectionEnable AND REAL_TO_BOOL(HMI_PAR_1._216) AND PstFlr.ProductionMode AND NOT TNK.DataOut.CipMode AND NOT TNK.DataOut.RinseMode;
	HMI_DOS_SS2P[SS2P_DOS_ModeProdFast].LampON		:= HMI_DOS_SS2P[SS2P_DOS_ModeProdFast].ON;

	IF EDGEPOS(VAR_DOS_ModeProduction) THEN //RESTORE SELECTION IN CASE OF POWER OFF
		HMI_DOS_SS2P[SS2P_DOS_ModeProdFast].ON := TRUE;
	END_IF

	//SS2P DOSER DRAIN
	HMI_DOS_SS2P[SS2P_DOS_ModeDrain].Visibility	:= TRUE;
	HMI_DOS_SS2P[SS2P_DOS_ModeDrain].Enable		:= VAR_DOS_SS2PSelectionEnable;
	HMI_DOS_SS2P[SS2P_DOS_ModeDrain].LampON		:= HMI_DOS_SS2P[SS2P_DOS_ModeDrain].ON;

	IF EDGEPOS(VAR_DOS_ModeDrain) THEN //RESTORE SELECTION IN CASE OF POWER OFF
		HMI_DOS_SS2P[SS2P_DOS_ModeDrain].ON := TRUE;
	END_IF

	//SS2P DOSER CIP
	HMI_DOS_SS2P[SS2P_DOS_ModeCip].Visibility	:= TRUE;
	HMI_DOS_SS2P[SS2P_DOS_ModeCip].Enable		:= VAR_DOS_SS2PSelectionEnable AND PstFlr.CipRunning AND NOT TNK.DataOut.ProdMode;
	HMI_DOS_SS2P[SS2P_DOS_ModeCip].LampON		:= HMI_DOS_SS2P[SS2P_DOS_ModeCip].ON;

	IF EDGEPOS(VAR_DOS_ModeCip) THEN //RESTORE SELECTION IN CASE OF POWER OFF
		HMI_DOS_SS2P[SS2P_DOS_ModeCip].ON := TRUE;
	END_IF

	//SS2P DOSER RINSE
	HMI_DOS_SS2P[SS2P_DOS_ModeRinse].Visibility	:= TRUE;
	HMI_DOS_SS2P[SS2P_DOS_ModeRinse].Enable		:= VAR_DOS_SS2PSelectionEnable AND NOT TNK.DataOut.ProdMode;
	HMI_DOS_SS2P[SS2P_DOS_ModeRinse].LampON		:= HMI_DOS_SS2P[SS2P_DOS_ModeRinse].ON;

	IF EDGEPOS(VAR_DOS_ModeRinse) THEN //RESTORE SELECTION IN CASE OF POWER OFF
		HMI_DOS_SS2P[SS2P_DOS_ModeRinse].ON := TRUE;
	END_IF

	//SS2P DOSER QUICK RINSE
	HMI_DOS_SS2P[SS2P_DOS_ModeQuickRinse].Visibility	:= FALSE;
	HMI_DOS_SS2P[SS2P_DOS_ModeQuickRinse].Enable		:= VAR_DOS_ModeWait;
	HMI_DOS_SS2P[SS2P_DOS_ModeQuickRinse].LampON		:= HMI_DOS_SS2P[SS2P_DOS_ModeQuickRinse].ON;

	//SS2P DOSER FAST RINSE
	HMI_DOS_SS2P[SS2P_DOS_ModeFastRinse].Visibility	:= FALSE;
	HMI_DOS_SS2P[SS2P_DOS_ModeFastRinse].Enable		:= VAR_DOS_ModeWait;
	HMI_DOS_SS2P[SS2P_DOS_ModeFastRinse].LampON		:= HMI_DOS_SS2P[SS2P_DOS_ModeFastRinse].ON;

//PB
	//Start Lifting Position button
	HMI_DOS_PB[PB_CmdLiftMotorStart].Visibility	:= TRUE;
	HMI_DOS_PB[PB_CmdLiftMotorStart].Enable		:= HMI_DOS_LiftPosition.Value <> 0 AND VAR_DOS_MotorEnable;
	HMI_DOS_PB[PB_CmdLiftMotorStart].LampON		:= HMI_DOS_PB[PB_CmdLiftMotorStart].ON;

	//Stop Lifting Position button
	HMI_DOS_PB[PB_CmdLiftMotorStop].Visibility	:= TRUE;
	HMI_DOS_PB[PB_CmdLiftMotorStop].Enable		:= HMI_DOS_LiftPosition.Value <> 0 AND VAR_DOS_MotorEnable;
	HMI_DOS_PB[PB_CmdLiftMotorStop].LampON		:= HMI_DOS_PB[PB_CmdLiftMotorStop].ON;

	//Manual Up Push Button
	HMI_DOS_PB[PB_DOS_Up].Visibility	:= TRUE;
	HMI_DOS_PB[PB_DOS_Up].LampON		:= HMI_DOS_PB[PB_DOS_Up].ON AND HMI_DOS_PB[PB_DOS_Up].Enable;

	//Manual Down Push Button
	HMI_DOS_PB[PB_DOS_Down].Visibility	:= TRUE;
	HMI_DOS_PB[PB_DOS_Down].LampON		:= HMI_DOS_PB[PB_DOS_Down].ON AND HMI_DOS_PB[PB_DOS_Down].Enable;

	//PB Mode Start
	HMI_DOS_PB[PB_CmdDosStart].Visibility				:= TRUE;
	HMI_DOS_PB[PB_CmdDosStart].Enable					:= (VAR_DOS_ModeWait OR VAR_DOS_SEQ.Mem.PBStartEnable);
	HMI_DOS_PB[PB_CmdDosStart].LampON					:= HMI_DOS_PB[PB_CmdDosStart].ON;
	HMI_DOS_PB[PB_CmdDosStart].Blink					:= VAR_DOS_ModeWait AND HMI_DOS_PB[PB_CmdDosStart].Enable AND (HMI_DOS_SS2P[SS2P_DOS_ModeProdFast].LampON OR HMI_DOS_SS2P[SS2P_DOS_ModeDrain].LampON OR HMI_DOS_SS2P[SS2P_DOS_ModeCip].LampON OR HMI_DOS_SS2P[SS2P_DOS_ModeRinse].LampON);

	//PB Mode Stop
	HMI_DOS_PB[PB_CmdDosStop].Visibility				:= TRUE;
	HMI_DOS_PB[PB_CmdDosStop].Enable					:= NOT VAR_DOS_ModeWait AND VAR_DOS_SEQ.Mem.PBStopEnable;
	HMI_DOS_PB[PB_CmdDosStop].LampON					:= HMI_DOS_PB[PB_CmdDosStop].ON;
	HMI_DOS_PB[PB_CmdDosStop].Blink						:= NOT VAR_DOS_ModeWait AND HMI_DOS_PB[PB_CmdDosStop].Enable;

	//PB Mode Skip
	HMI_DOS_PB[PB_CmdDosSkip].Visibility				:= FALSE;
	HMI_DOS_PB[PB_CmdDosSkip].Enable					:= NOT VAR_DOS_ModeWait;
	HMI_DOS_PB[PB_CmdDosSkip].LampON					:= HMI_DOS_PB[PB_CmdDosSkip].ON;

	//PB Mode Pause
	HMI_DOS_PB[PB_CmdDosPause].Visibility				:= FALSE;
	HMI_DOS_PB[PB_CmdDosPause].Enable					:= NOT VAR_DOS_ModeWait;
	HMI_DOS_PB[PB_CmdDosPause].LampON					:= HMI_DOS_PB[PB_CmdDosPause].ON;

	//PB Mode Abort
	HMI_DOS_PB[PB_CmdDosAbort].Visibility				:= TRUE;
	HMI_DOS_PB[PB_CmdDosAbort].Enable					:= NOT VAR_DOS_ModeWait AND VAR_DOS_SEQ.Mem.PBAbortEnable;
	HMI_DOS_PB[PB_CmdDosAbort].LampON					:= HMI_DOS_PB[PB_CmdDosAbort].ON;

	//SS3P
	HMI_DOS_SS3P[SS3P_DOS_FillingValveOpen].Visibility	:= TRUE;
	HMI_DOS_SS3P[SS3P_DOS_FillingValveOpen].Enable		:= HMI_SS2P[SS2P_HMI_SelEnable].ON AND DOS.DataOut.ProdMode;
	HMI_DOS_SS3P[SS3P_DOS_FillingValveOpen].LampON		:= IO_210CPF.DO_Opened;

	//STATUS BAR
	HMI_DOS_State.Sequencer.TextBar[0].Visibility	:= TRUE;
	HMI_DOS_State.Sequencer.TextBar[0].IndexNr		:= FB_DOS_SEQ.IN_Step;
	HMI_DOS_State.Sequencer.TextBar[0].IndexText	:= FB_DOS_SEQ.OUT_HMI_ID;

	HMI_DOS_State.Sequencer.TextBar[1].Visibility	:= FALSE;
	HMI_DOS_State.Sequencer.TextBar[1].IndexNr		:= 0;
	HMI_DOS_State.Sequencer.TextBar[1].IndexText	:= 0;

	// HMI VARIABLES
	IF (VAR_DOS_ModeProduction OR VAR_DOS_FMDProductionFillerOnly OR (VAR_DOS_ModeWait AND (HMI_DOS_LiftPosition.Value = 1))) THEN
		HMI_DOS_DosingVolumeSp :=  HMI_PAR_1._215;
	ELSIF ((VAR_DOS_ModeCip OR VAR_DOS_ModeRinse) OR (VAR_DOS_ModeWait AND (HMI_DOS_LiftPosition.Value = 3))) THEN
		HMI_DOS_DosingVolumeSp := VAR_DOS_Lift_State.CmdCipHeight.Sp;
	ELSIF ((VAR_DOS_ModeCop AND COP.DataOut.DoserPositioningReq) OR (VAR_DOS_ModeWait AND (HMI_DOS_LiftPosition.Value = 2))) THEN
		HMI_DOS_DosingVolumeSp := 0; ////High sensor _215DSF, SP in mm in COP
	ELSE
		HMI_DOS_DosingVolumeSp := 0;
	END_IF

	HMI_DOS_DosingVolumePv							:= VAR_DOS_MMF205.PosActual[ml];
	HMI_DOS_Bypass_State.Active						:= GNS.DataOut.DosByPassed;
	HMI_DOS_Bypass_State.Fault						:= GNS.DataOut.DosByPassAlarm;
	HMI_DOS_PstFlrEndProductionReq					:= PstFlr.EndProductionReq; //rma106
	HMI_DOS_ProdEndNecessaryBottle					:= REAL_TO_DINT(VAR_DOS_ProdEndNecessaryBottle);

	//INFO BOX:STEPS
	HMI_DOS_State.Sequencer.InfoBox[0].Visibility			:= FB_DOS_SEQ.OUT_StepTimePr_T>0 OR FB_DOS_SEQ.OUT_StepTimePr_TON>0;
	HMI_DOS_State.Sequencer.InfoBox[0].IndexText			:= '@Lbl_Step@ time';
	HMI_DOS_State.Sequencer.InfoBox[0].Unit					:= 0;
	HMI_DOS_State.Sequencer.InfoBox[0].ProgressVisibility	:= TRUE;
	HMI_DOS_State.Sequencer.InfoBox[0].Progress				:= UINT_TO_REAL(FB_DOS_SEQ.OUT_StepProgressiveTime);
	IF FB_DOS_SEQ.OUT_StepTimePr_T>0 THEN
		HMI_DOS_State.Sequencer.InfoBox[0].Preset			:= UINT_TO_REAL(FB_DOS_SEQ.OUT_StepTimePr_T);
	ELSE
		HMI_DOS_State.Sequencer.InfoBox[0].Preset			:= UINT_TO_REAL(FB_DOS_SEQ.OUT_StepTimePr_TON);
	END_IF
	IF FB_DOS_SEQ.OUT_StepTimePr_T>0 THEN
		HMI_DOS_State.Sequencer.InfoBox[0].Actual			:= UINT_TO_REAL(FB_DOS_SEQ.OUT_StepTimeCV_T);
	ELSE
		HMI_DOS_State.Sequencer.InfoBox[0].Actual			:= UINT_TO_REAL(FB_DOS_SEQ.OUT_StepTimeCV_TON);
	END_IF
	//SIGNALS STATE:PRODUCTION
	//DigitalIn[0]
	HMI_DOS_State.Signals.DigitalIn[1].Visibility	:= TRUE;
	HMI_DOS_State.Signals.DigitalIn[1].LampState	:= PstFlr.ProductionMode;
	HMI_DOS_State.Signals.DigitalIn[1].Description	:= '@External Signal Production Enable';

	HMI_DOS_State.Signals.DigitalOut[1].Visibility	:= TRUE;
	HMI_DOS_State.Signals.DigitalOut[1].LampState	:= VAR_DOS_ModeWait;
	HMI_DOS_State.Signals.DigitalOut[1].Description	:= '@Filler Signal Production Enable';

	//SIGNALS STATE:DRAIN
	//DigitalIn[1]
	HMI_DOS_State.Signals.DigitalIn[2].Visibility	:= TRUE;
	HMI_DOS_State.Signals.DigitalIn[2].LampState	:= TRUE;
	HMI_DOS_State.Signals.DigitalIn[2].Description	:= '@External Signal Drain Enable';

	HMI_DOS_State.Signals.DigitalOut[2].Visibility	:= TRUE;
	HMI_DOS_State.Signals.DigitalOut[2].LampState	:= VAR_DOS_ModeWait;
	HMI_DOS_State.Signals.DigitalOut[2].Description	:= '@Filler Signal Drain Enable';

	//SIGNALS STATE:Alive
	//DigitalIn[2]
	HMI_DOS_State.Signals.DigitalIn[3].Visibility	:= FALSE;
	HMI_DOS_State.Signals.DigitalIn[3].LampState	:= FALSE;
	HMI_DOS_State.Signals.DigitalIn[3].Description	:= '@Alive';

	HMI_DOS_State.Signals.DigitalOut[3].Visibility	:= FALSE;
	HMI_DOS_State.Signals.DigitalOut[3].LampState	:= FALSE;
	HMI_DOS_State.Signals.DigitalOut[3].Description	:= '@Alive';

	//SIGNALS STATE:CLEANING
	//DigitalIn[3]
	HMI_DOS_State.Signals.DigitalIn[4].Visibility	:= TRUE;
	HMI_DOS_State.Signals.DigitalIn[4].LampState	:= PstFlr.CipRunning;
	HMI_DOS_State.Signals.DigitalIn[4].Description	:= '@External Signal CIP Enable';

	HMI_DOS_State.Signals.DigitalOut[4].Visibility	:= TRUE;
	HMI_DOS_State.Signals.DigitalOut[4].LampState	:= VAR_DOS_ModeWait;
	HMI_DOS_State.Signals.DigitalOut[4].Description	:= '@Filler Signal CIP Enable';

	//SIGNALS STATE:RINSE
	//DigitalIn[4]
	HMI_DOS_State.Signals.DigitalIn[5].Visibility	:= TRUE;
	HMI_DOS_State.Signals.DigitalIn[5].LampState	:= PstFlr.RinseMode;
	HMI_DOS_State.Signals.DigitalIn[5].Description	:= '@External Signal Rinse Enable';

	HMI_DOS_State.Signals.DigitalOut[5].Visibility	:= TRUE;
	HMI_DOS_State.Signals.DigitalOut[5].LampState	:= VAR_DOS_ModeWait;
	HMI_DOS_State.Signals.DigitalOut[5].Description	:= '@Filler Signal Rinse Enable';

END_ACTION
```

#### DOS_Alarm.st
```iecst
ACTION DOS_Alarm:
	//PULP DOSER HEMA ALARM
	ALR[3021].Active	:= VAR_DOS_AVJ_ValveFault;
	ALR[3001].Active	:= LTJ[203].OUT_Alarm;
	ALR[3002].Active	:= TTJ[203].OUT_Alarm;
	ALR[3003].Active	:= MMJ[201].OUT_OverloadFault;
	ALR[3005].Active	:= MMJ[201].OUT_DriveFault;
	ALR[3006].Active	:= MMJ[201].OUT_IsolatedFault;
	ALR[3008].Active;//FAN SHAKER MOTOR
	ALR[3009].Active;//FAN SHAKER MOTOR
	ALR[3013].Active	:= VAR_DOS_NoBotNoFillPressureFault;
	ALR[3014].Active	:= VAR_DOS_NoBotNoFillPressureLow;
	ALR[3017].Active	:= VAR_DOS_WaterTemperatureTooLow;
	ALR[3018].Active	:= VAR_DOS_WaterTemperatureTooHigh;
	ALR[3019].Active	:= VAR_DOS_StepProdLowLevel;
	//ALR[3020].Active	:= VAR_DOS_TankTooFull;
	ALR[3024].Active; //ZERO POSITION NOT FOUND
	ALR[3025].Active := MMF[205].OUT_OverloadFault;
	ALR[3027].Active := _205MEF.OUT_Alarm;
	ALR[3028].Active := MMF[205].OUT_DriveFault;
	ALR[3029].Active := MMF[206].OUT_OverloadFault;
	ALR[3031].Active := FALSE; // leo _206MEF.OUT_Alarm;
	ALR[3032].Active := MMF[206].OUT_DriveFault;
	ALR[3041].Active := PPJ[202].OUT_OverloadFault;
	ALR[3043].Active := PPJ[202].OUT_DriveFault;
	ALR[3044].Active := PPJ[202].OUT_IsolatedFault;
	ALR[3048].Active := VAR_DOS_CleanArmCopPosFault;
	ALR[3051].Active := (VAR_DOS_ModeProduction OR VAR_DOS_ModeCip OR VAR_DOS_ModeDrain OR VAR_DOS_ModeRinse) AND VAR_DOS_CleanArmCopPos;//Quick stop se viene alzata richiesta con Arm cleaning inserito
	ALR[3010].Active := VAR_DOS_StepCamPosInProgress; //OR (VAR_DOS_BypassRequest; //Bypass Request -> Machine empty + Normal Stop
	ALR[3015].Active := GNS.DataOut.DosByPassAlarm; //Error bypass -> Critical Stop
	ALR[3016].Active := VAR_DOS_StepMotorization; //Motorization Check
	ALR[3011].Active := HMI_DOS_SS3P[SS3P_DOS_FillingValveOpen].Visibility AND NOT HMI_DOS_SS3P[SS3P_DOS_FillingValveOpen].Auto;
	ALR[3057].Active := VAR_DOS_EndProdStopContainer;
	ALR[3058].Active := VAR_DOS_SEQ.Mem.ContainersStop AND VAR_DOS_ModeProduction;

	ALR[3022].Active := LSJ[202].OUT;

	TON_DosRunFbk[0].IN := MMF[205].OUT_InOperation AND NOT TON_DosRunFbk[0].Q;
	TON_DosRunFbk[0].PT := t#3s;
	TON_DosRunFbk[0]();

	TON_DosRunFbk[1].IN := MMF[206].OUT_InOperation AND NOT TON_DosRunFbk[1].Q;
	TON_DosRunFbk[1].PT := t#3s;
	TON_DosRunFbk[1]();

	//MMF205
	IF EDGEPOS(TON_DosRunFbk[0].IN) THEN
		VAR_MMF205PositionSave := _205MEF.OUT_ActValue;
		VAR_MMF205Down 			:=	MMF[205].IN_Reverse;
	ELSIF EDGEPOS(TON_DosRunFbk[0].Q) THEN
		IF VAR_MMF205Down AND (_205MEF.OUT_ActValue >= VAR_MMF205PositionSave) THEN
			VAR_DOS_LiftMMF205SeqMem.LiftMotor.RunFbkAlr := TRUE;
		ELSIF NOT VAR_MMF205Down AND (_205MEF.OUT_ActValue <= (VAR_MMF205PositionSave)) THEN
			VAR_DOS_LiftMMF205SeqMem.LiftMotor.RunFbkAlr := TRUE;
		END_IF
	END_IF
	IF AID.DataOut.Reset THEN
		VAR_DOS_LiftMMF205SeqMem.LiftMotor.RunFbkAlr := FALSE;
	END_IF
	ALR[939].Active 	:= VAR_DOS_LiftMMF205SeqMem.LiftMotor.RunFbkAlr; // New alarm to check the movement

	//MMF206
	IF EDGEPOS(TON_DosRunFbk[1].IN) THEN
		VAR_MMF206PositionSave := _206MEF.OUT_ActValue;
		VAR_MMF206Down 			:= MMF[206].IN_Reverse;
	ELSIF EDGEPOS(TON_DosRunFbk[1].Q) THEN
		IF VAR_MMF206Down AND (_206MEF.OUT_ActValue >= VAR_MMF206PositionSave) THEN
			VAR_DOS_LiftMMF206SeqMem.LiftMotor.RunFbkAlr := TRUE;
		ELSIF NOT VAR_MMF206Down AND (_206MEF.OUT_ActValue <= (VAR_MMF206PositionSave)) THEN
			VAR_DOS_LiftMMF206SeqMem.LiftMotor.RunFbkAlr := TRUE;
		END_IF
	END_IF
	IF AID.DataOut.Reset THEN
		VAR_DOS_LiftMMF206SeqMem.LiftMotor.RunFbkAlr := FALSE;
	END_IF
	ALR[941].Active 	:= VAR_DOS_LiftMMF206SeqMem.LiftMotor.RunFbkAlr; // New alarm to check the movement

	//*******************************************************
	TON_DosPositionCheck[0].IN := MMF[205].OUT_InOperation;
	TON_DosPositionCheck[0].PT := t#3s;
	TON_DosPositionCheck[0]();

	TON_DosPositionCheck[1].IN := MMF[206].OUT_InOperation;
	TON_DosPositionCheck[1].PT := t#3s;
	TON_DosPositionCheck[1]();

	//MMF205
	IF EDGEPOS(TON_DosPositionCheck[0].IN) THEN
		VAR_OldMMF205Position := _205MEF.OUT_ActValue;
		VAR_MMF205DirectionReverse := MMF[205].IN_Reverse;
	END_IF

	IF TON_DosPositionCheck[0].Q THEN
		IF VAR_MMF205DirectionReverse THEN
			IF _205MEF.OUT_ActValue > VAR_OldMMF205Position THEN
				VAR_DOS_LiftMMF205SeqMem.LiftMotor.DirectionAlr := TRUE;
			END_IF
		ELSIF _205MEF.OUT_ActValue < VAR_OldMMF205Position THEN
			VAR_DOS_LiftMMF205SeqMem.LiftMotor.DirectionAlr := TRUE;
		END_IF
		TON_DosPositionCheck[0](IN := FALSE);
		VAR_OldMMF205Position := _205MEF.OUT_ActValue;
	ELSIF AID.DataOut.Reset THEN
		VAR_DOS_LiftMMF205SeqMem.LiftMotor.DirectionAlr := FALSE;
	END_IF

	IF EDGEPOS(TON_DosPositionCheck[1].IN) THEN
		VAR_OldMMF206Position := _206MEF.OUT_ActValue;
		VAR_MMF206DirectionReverse := MMF[206].IN_Reverse;
	END_IF
	ALR[940].Active 	:= VAR_DOS_LiftMMF205SeqMem.LiftMotor.DirectionAlr;

	//MMF206
	IF TON_DosPositionCheck[1].Q THEN
		IF VAR_MMF206DirectionReverse THEN
			IF _206MEF.OUT_ActValue > VAR_OldMMF206Position THEN
				VAR_DOS_LiftMMF206SeqMem.LiftMotor.DirectionAlr := TRUE;
			END_IF
		ELSIF _206MEF.OUT_ActValue < VAR_OldMMF206Position THEN
			VAR_DOS_LiftMMF206SeqMem.LiftMotor.DirectionAlr := TRUE;
		END_IF
		TON_DosPositionCheck[1](IN := FALSE);
		VAR_OldMMF206Position := _206MEF.OUT_ActValue;
	ELSIF AID.DataOut.Reset THEN
		VAR_DOS_LiftMMF206SeqMem.LiftMotor.DirectionAlr := FALSE;
	END_IF
	ALR[942].Active 	:= VAR_DOS_LiftMMF206SeqMem.LiftMotor.DirectionAlr;
END_ACTION
```

#### DOS_AlarmFlavor.st
```iecst
ACTION DOS_AlarmFlavor:
	//FLAVOR DOSER ALARM
	ALR[3100].ActionEn := TRUE;
	IF (NOT DosFlr.Fault)
		OR (DosFlr.OutOfService AND FlrDos.AromePodReq AND TNK.DataOut.ProdMode)
		OR (NOT DosFlr.OutOfService AND NOT FlrDos.AromePodReq AND TNK.DataOut.ProdMode)  THEN
		ALR[3100].Active := TRUE;
	ELSE
		ALR[3100].Active := FALSE;
	END_IF

	ALR[3101].Active	:= NOT DosFlr.ContainerBlock OR NOT DosFlr.ProdReady;
	ALR[3102].ActionEn 	:= TNK.DataOut.ProdMode OR TNK.DataOut.CipMode;
	ALR[3102].Active	:= NOT IO_DOS_OverloadOk.DI_Input;

	//V4.A.A.1.6.13
	ALR[3103].Active	:= DosFlr.CipReady AND NOT DosFlr.CipRunning;
	ALR[3104].Active 	:= DosFlr.PrimingCycleProgress;
	ALR[3105].Active	:= DosFlr.SampleCycleInProgress;
	ALR[3106].Active 	:= DosFlr.SettingCycleInProgress;
	ALR[3107].Active 	:= DosFlr.Positioning (*AND NOT FlrDos.PositioningDone*);

END_ACTION
```

#### DOS_Hardware_CFG.st
```iecst
ACTION DOS_Hardware_CFG:
	(***** VALVES *****)
	AVJ[201].IN_ConfigPresent				:= TRUE;
	AVJ[201].IN_ConfigType 					:= 0;
	AVJ[201].IN_Simulation 					:= FALSE;
	AVJ[201].IN_ConfigPositionSensorOpened 	:= TRUE;
	AVJ[201].IN_ConfigPositionSensorClosed 	:= TRUE;
	AVJ[201].IN_StrokeTime 					:= T#5s;

	AVJ[210].IN_ConfigPresent				:= TRUE;
	AVJ[210].IN_ConfigType 					:= 0;
	AVJ[210].IN_Simulation 					:= FALSE;
	AVJ[210].IN_ConfigPositionSensorOpened 	:= TRUE;
	AVJ[210].IN_ConfigPositionSensorClosed 	:= TRUE;
	AVJ[210].IN_StrokeTime 					:= T#5s;

	AVJ[211].IN_ConfigPresent				:= TRUE;
	AVJ[211].IN_ConfigType 					:= 0;
	AVJ[211].IN_Simulation 					:= FALSE;
	AVJ[211].IN_ConfigPositionSensorOpened 	:= TRUE;
	AVJ[211].IN_ConfigPositionSensorClosed 	:= TRUE;
	AVJ[211].IN_StrokeTime 					:= T#5s;

	AVJ[212].IN_ConfigPresent				:= FALSE;
	AVJ[212].IN_ConfigType 					:= 0;
	AVJ[212].IN_Simulation 					:= FALSE;
	AVJ[212].IN_ConfigPositionSensorOpened 	:= TRUE;
	AVJ[212].IN_ConfigPositionSensorClosed 	:= TRUE;
	AVJ[212].IN_StrokeTime 					:= T#5s;

	AVJ[215].IN_ConfigPresent				:= TRUE;
	AVJ[215].IN_ConfigType 					:= 0;
	AVJ[215].IN_ConfigNormallyOpen			:= FALSE;
	AVJ[215].IN_Simulation 					:= FALSE;
	AVJ[215].IN_ConfigPositionSensorOpened 	:= TRUE;
	AVJ[215].IN_ConfigPositionSensorClosed 	:= TRUE;
	AVJ[215].IN_StrokeTime 					:= T#5s;

	AVJ[216].IN_ConfigPresent				:= TRUE;
	AVJ[216].IN_ConfigType 					:= 0;
	AVJ[216].IN_Simulation 					:= FALSE;
	AVJ[216].IN_ConfigPositionSensorOpened 	:= TRUE;
	AVJ[216].IN_ConfigPositionSensorClosed 	:= TRUE;
	AVJ[216].IN_StrokeTime 					:= T#5s;

	AVJ[217].IN_ConfigPresent				:= TRUE;
	AVJ[217].IN_ConfigType 					:= 0;
	AVJ[217].IN_Simulation 					:= FALSE;
	AVJ[217].IN_ConfigPositionSensorOpened 	:= FALSE;
	AVJ[217].IN_ConfigPositionSensorClosed 	:= FALSE;
	AVJ[217].IN_StrokeTime 					:= T#5s;

	AVJ[218].IN_ConfigPresent				:= FALSE;
	AVJ[218].IN_ConfigType 					:= 0;
	AVJ[218].IN_Simulation 					:= FALSE;
	AVJ[218].IN_ConfigPositionSensorOpened 	:= TRUE;
	AVJ[218].IN_ConfigPositionSensorClosed 	:= TRUE;
	AVJ[218].IN_StrokeTime 					:= T#5s;

	AVJ[221].IN_ConfigPresent				:= FALSE;
	AVJ[221].IN_ConfigType 					:= 0;
	AVJ[221].IN_ConfigNormallyOpen			:= TRUE;
	AVJ[221].IN_Simulation 					:= FALSE;
	AVJ[221].IN_ConfigPositionSensorOpened 	:= TRUE;
	AVJ[221].IN_ConfigPositionSensorClosed 	:= TRUE;
	AVJ[221].IN_StrokeTime 					:= T#5s;

	AVJ[230].IN_ConfigPresent				:= CFG_Par.Doser.RecoverySkid;
	AVJ[230].IN_ConfigType 					:= 0;
	AVJ[230].IN_ConfigNormallyOpen			:= FALSE;
	AVJ[230].IN_Simulation 					:= FALSE;
	AVJ[230].IN_ConfigPositionSensorOpened 	:= TRUE;
	AVJ[230].IN_ConfigPositionSensorClosed 	:= TRUE;
	AVJ[230].IN_StrokeTime 					:= T#5s;

	AVJ[231].IN_ConfigPresent				:= CFG_Par.Doser.RecoverySkid;
	AVJ[231].IN_ConfigType 					:= 0;
	AVJ[231].IN_ConfigNormallyOpen			:= FALSE;
	AVJ[231].IN_Simulation 					:= FALSE;
	AVJ[231].IN_ConfigPositionSensorOpened 	:= TRUE;
	AVJ[231].IN_ConfigPositionSensorClosed 	:= TRUE;
	AVJ[231].IN_StrokeTime 					:= T#5s;

	AVJ[232].IN_ConfigPresent				:= CFG_Par.Doser.RecoverySkid;
	AVJ[232].IN_ConfigType 					:= 0;
	AVJ[232].IN_ConfigNormallyOpen			:= FALSE;
	AVJ[232].IN_Simulation 					:= FALSE;
	AVJ[232].IN_ConfigPositionSensorOpened 	:= TRUE;
	AVJ[232].IN_ConfigPositionSensorClosed 	:= TRUE;
	AVJ[232].IN_StrokeTime 					:= T#5s;

	AVJ[233].IN_ConfigPresent				:= CFG_Par.Doser.RecoverySkid;
	AVJ[233].IN_ConfigType 					:= 0;
	AVJ[233].IN_ConfigNormallyOpen			:= FALSE;
	AVJ[233].IN_Simulation 					:= FALSE;
	AVJ[233].IN_ConfigPositionSensorOpened 	:= TRUE;
	AVJ[233].IN_ConfigPositionSensorClosed 	:= TRUE;
	AVJ[233].IN_StrokeTime 					:= T#5s;

	AVJ[234].IN_ConfigPresent				:= CFG_Par.Doser.RecoverySkid;
	AVJ[234].IN_ConfigType 					:= 0;
	AVJ[234].IN_ConfigNormallyOpen			:= FALSE;
	AVJ[234].IN_Simulation 					:= FALSE;
	AVJ[234].IN_ConfigPositionSensorOpened 	:= TRUE;
	AVJ[234].IN_ConfigPositionSensorClosed 	:= TRUE;
	AVJ[234].IN_StrokeTime 					:= T#5s;

	AVJ[235].IN_ConfigPresent				:= CFG_Par.Doser.RecoverySkid;
	AVJ[235].IN_ConfigType 					:= 0;
	AVJ[235].IN_ConfigNormallyOpen			:= FALSE;
	AVJ[235].IN_Simulation 					:= FALSE;
	AVJ[235].IN_ConfigPositionSensorOpened 	:= TRUE;
	AVJ[235].IN_ConfigPositionSensorClosed 	:= TRUE;
	AVJ[235].IN_StrokeTime 					:= T#5s;

	RVJ[201].IN_ConfigPresent 				:= FALSE;
	RVJ[201].IN_Simulation 					:= FALSE;
	RVJ[201].IN_ConfigPositionSensorOpened 	:= FALSE;
	RVJ[201].IN_ConfigPositionSensorClosed 	:= FALSE;
	RVJ[201].IN_ConfigPositionAnalogFBK 	:= FALSE;
	RVJ[201].IN_StrokeTime 					:= t#3s;
	RVJ[201].IN_ConfigNormallyOpen 			:= FALSE;

	(***** MOTORS *****)
	PPJ[202].IN_ConfigPresent				:= CFG_Par.Doser.Present;
	PPJ[202].IN_Reverse						:= FALSE;
	PPJ[202].IN_ManEn						:= TRUE;
	PPJ[202].IN_FrequencyMin				:= 0.0;
	PPJ[202].IN_FrequencyMax				:= 60.0;

	PPJ203.IN_ConfigPresent					:= FALSE;
	PPJ203.IN_ManEn							:= TRUE;
	PPJ203.IN_Simulation 					:= FALSE;

	MMJ[201].IN_ConfigPresent				:= CFG_Par.Doser.Present;
	MMJ[201].IN_Reverse						:= FALSE;
	MMJ[201].IN_ManEn						:= TRUE;
	MMJ[202].IN_FrequencyMin				:= 0.0;
	MMJ[202].IN_FrequencyMax				:= 100.0;

	MMF[205].IN_ConfigPresent				:= CFG_Par.Doser.Present;
	MMF[205].IN_ManEn						:= TRUE;
	MMF[205].IN_FrequencyMin				:= 0.0;
	MMF[205].IN_FrequencyMax				:= 60.0;

	MMF[206].IN_ConfigPresent				:= CFG_Par.Doser.Present;
	MMF[206].IN_ManEn						:= TRUE;
	MMF[206].IN_FrequencyMin				:= 0.0;
	MMF[206].IN_FrequencyMax				:= 60.0;

	(***** ANALOG *****)
	LTJ[203].IN_ConfigPresent				:= CFG_Par.Doser.Present;
	LTJ[203].IN_Simulation					:= FALSE;
	LTJ[203].IN_0_20mA						:= TRUE;
	LTJ[203].IN_ScaleLOW					:= 0;
	LTJ[203].IN_ScaleHIGH					:= 100; //%
	LTJ[203].IN_MaskEn						:= TRUE;
	LTJ[203].IN_ConfigPopup					:= TRUE;
	LTJ[203].IN_CompareMode					:= VAR_DOS_SEQ.Device.LTJ203.CMP;

	TTJ[203].IN_ConfigPresent				:= CFG_Par.Doser.Present;
	TTJ[203].IN_Simulation					:= FALSE;
	TTJ[203].IN_0_20mA						:= TRUE;
	TTJ[203].IN_ScaleLOW					:= 0.0;
	TTJ[203].IN_ScaleHIGH					:= 100.0;
	TTJ[203].IN_MaskEn						:= TRUE;
	TTJ[203].IN_ConfigPopup					:= TRUE;
	TTJ[203].IN_CompareMode					:= VAR_DOS_SEQ.Device.TTJ203.CMP;

	_210PTF.IN_ConfigPresent 				:= CFG_Par.Doser.Present;
	_210PTF.IN_OffDelay;
	_210PTF.IN_OnDelay;

	//FILIPPO
	_205MEF.IN_ConfigPresent					:= TRUE;
	_205MEF.IN_Simulation						:= FALSE;
	_205MEF.IN_0_20mA							:= TRUE;
	_205MEF.IN_ScaleLOW							:= 0.0;
	_205MEF.IN_ScaleHIGH						:= 680.0; //Probe Lenght datasheet
	_205MEF.IN_AlarmEn							:= TRUE;
	_205MEF.IN_MinDev							:= 1.0; //[mm]
	_205MEF.IN_MaxDev							:= 1.0; //[mm]
	_205MEF.IN_WaitDelay						:= t#100ms;
	_205MEF.IN_HighLimitEn						:= TRUE;
	_205MEF.IN_HighLimitSP						:= 200.0;
	_205MEF.IN_HighLimitHyst					:= 0.0 ;
	_205MEF.IN_HighLimitDelay					:= t#100ms;
	_205MEF.IN_LowLimitEn						:= TRUE;
	_205MEF.IN_LowLimitSP						:= 8.0;
	_205MEF.IN_LowLimitHyst						:= 0.0;
	_205MEF.IN_LowLimitDelay					:= t#100ms;
	_205MEF.IN_Direct_Inverse					:= TRUE; //FALSE = Direct - TRUE = Inverse
	//_205MEF.IN_Delta							:= -308.0; //[mm] Delta Value for Real Component Height (always added to the Probe Value) To define in test with ADJ

	//_206MEF
	_206MEF.IN_ConfigPresent					:= TRUE;
	_206MEF.IN_Simulation						:= FALSE;
	_206MEF.IN_0_20mA							:= TRUE;
	_206MEF.IN_ScaleLOW							:= 0.0;
	_206MEF.IN_ScaleHIGH						:= 680.0; //Probe Lenght datasheet
	_206MEF.IN_AlarmEn							:= TRUE;
	_206MEF.IN_MinDev							:= 1.0; //[mm]
	_206MEF.IN_MaxDev							:= 1.0; //[mm]
	_206MEF.IN_WaitDelay						:= t#100ms;
	_206MEF.IN_HighLimitEn						:= TRUE;
	_206MEF.IN_HighLimitSP						:= 200.0;
	_206MEF.IN_HighLimitHyst					:= 0.0 ;
	_206MEF.IN_HighLimitDelay					:= t#100ms;
	_206MEF.IN_LowLimitEn						:= TRUE;
	_206MEF.IN_LowLimitSP						:= 8.0;
	_206MEF.IN_LowLimitHyst						:= 0.0;
	_206MEF.IN_LowLimitDelay					:= t#100ms;
	_206MEF.IN_Direct_Inverse					:= TRUE; //FALSE = Direct - TRUE = Inverse
	//_206MEF.IN_Delta							:= -310.0; //[mm] Delta Value for Real Component Height (always added to the Probe Value) To define in test with ADJ

	(***** DIGITAL *****) //FILIPPO
	_215DSF.IN_ConfigPresent 					:= TRUE;
	_216DSF.IN_ConfigPresent 					:= TRUE;
	_217DSF.IN_ConfigPresent 					:= TRUE;
	_210DSX.IN_ConfigPresent 					:= TRUE;
	_211DSX.IN_ConfigPresent 					:= TRUE;

	_212DSF.IN_ConfigPresent 					:= TRUE;
	_213DSF.IN_ConfigPresent 					:= TRUE;

	_211CPF.IN_ConfigPresent					:= TRUE;

	LSJ200L.IN_ConfigPresent					:= CFG_Par.Doser.RecoverySkid;
	LSJ200M.IN_ConfigPresent					:= CFG_Par.Doser.RecoverySkid;
	LSJ200H.IN_ConfigPresent					:= CFG_Par.Doser.RecoverySkid;
	LSJ[201].IN_ConfigPresent					:= CFG_Par.Doser.RecoverySkid;
	LSJ[202].IN_ConfigPresent					:= CFG_Par.Doser.RecoverySkid;
	FSJ[201].IN_ConfigPresent					:= CFG_Par.Doser.RecoverySkid;
	FSJ[202].IN_ConfigPresent					:= CFG_Par.Doser.RecoverySkid;

END_ACTION
```

Listed in the project but not available here: Logical/00_AID/AID/0010_Miscellany, Logical/00_AID/AID/0030_Beacon, Logical/00_AID/AID/0040_PbLight, Logical/00_AID/IO/IO_J.var, Logical/00_AID/Modules/Module_Types/DAQ_Global.typ, Logical/00_AID/Modules/Module_Types/CTP_Global.typ, Logical/00_AID/Modules/Module_Variables/DAQ_Global.var, Logical/00_AID/Modules/Module_Variables/CTP_Global.var, Logical/00_AID/Libraries/Sidel_Libraries/Sidel/FB_VFD_DataRead.st, Logical/00_AID/Libraries/Sidel_Libraries/Sidel_Obj/Dosing_Obj.st, Logical/02_HMI/HMI/HMI_Loading_Action/HMI_DAQ_Loading.st, Logical/02_HMI/HMI/HMI_Loading_Action/HMI_CTP_Loading.st, Logical/02_HMI/HMI/HMI_Loading_Action/HMI_DOS_Loading.st, Logical/02_HMI/HMI_Types/HMI_CTP.typ, Logical/02_HMI/HMI_Types/HMI_DAQ.typ, Logical/02_HMI/HMI_Types/HMI_DOS.typ, Logical/02_HMI/HMI_Variables/HMI_DOS.var, Logical/02_HMI/HMI_Variables/HMI_CTP.var, Logical/02_HMI/HMI_Variables/HMI_DAQ.var, Logical/02_HMI/HMI_Variables/HMI_J.var
